// TIA Portal V21 export
TYPE "TypeC0"
   STRUCT
      Heated_Lines_Enabled : Bool;   // true = Heated line/s are enabled
      Insulation_Monitor_Enabled : Bool;   // true = Insulation monitor is enabled
      Power_L2_Disabled : Bool;   // true = Power L2 is disabled
      Power_L4_Disabled : Bool;   // true = Power L4 is disabled
      Power_L6_Disabled : Bool;   // true = Power L6 is disabled
      Safety_Z2_Disabled : Bool;   // true = Safety Z2 is disabled
      Safety_Z4_Disabled : Bool;   // true = Safety Z4 is disabled
      Safety_Z6_Disabled : Bool;   // true = Safety Z6 is disabled
      Safety_Z8_Disabled : Bool;   // true = Safety Z8 is disabled
      HWCombiNumber : Int;   // PLC hardware combination number
   END_STRUCT;
END_TYPE
